// TIA Portal V18 export
FUNCTION_BLOCK "Slow_inc_quick_drop"   // FB50, FBD
{ S7_Optimized_Access := 'TRUE' }
VERSION : 0.1
// stored: AutoNumber true, IsIECCheckEnabled false, IsRetainMemResEnabled false, MemoryReserve 100, SetENOAutomatically false, UDAEnableTagReadback false
   VAR_INPUT
      ALLOWED : Bool;
      max_v : Real;
      sec_to_max_v : Real;
      req_v : Real;
   END_VAR
   VAR_OUTPUT
      speed : Real;
      er_set { ExternalAccessible := 'False'; ExternalVisible := 'False'; ExternalWritable := 'False'} : Bool;
      wsER : WString;
   END_VAR
   VAR
      accel_v_p_sec : Real;
      accel_per_cycle : Real;
      cycle_time_sec : Real := 0.01;
   END_VAR
BEGIN

REGION Network 2 (SCL)


   #er_set :=  "_MAIN_DB".CLOCK_S_P_SCAN <= 0 OR #sec_to_max_v <=0 ;
   IF #er_set THEN
       #wsER := WSTRING#'ошибка модуля ускорения';
   ELSE
       #wsER := WSTRING#'';
   END_IF;
END_REGION

REGION Network 3 (SCL)
   IF NOT #er_set THEN
       #accel_v_p_sec := #max_v / #sec_to_max_v;
       #accel_per_cycle := #accel_v_p_sec * "_MAIN_DB".CLOCK_S_P_SCAN;
   ELSE
       #accel_per_cycle := 0.0001;
   END_IF;
END_REGION

REGION Network 4 (SCL)
   IF #ALLOWED THEN
       IF NOT #er_set THEN
           IF #req_v > #speed THEN
               #speed := MIN(IN1 := #speed + #accel_per_cycle, IN2 := #req_v);
           ELSIF #req_v < #speed THEN
               #speed := MAX(IN1 := #speed - #accel_per_cycle, IN2 := #req_v);
           END_IF;

       ELSE
           #speed := 0;
       END_IF;
   ELSE
       #speed := 0;
   END_IF;
END_REGION
END_FUNCTION_BLOCK
